// TIA Portal V17 export
// export: Created 2025-03-05T08:00:56.2368358Z, ExportSetting WithDefaults, DisplayName Totally Integrated Automation Portal, DisplayVersion V17 Update 8, DisplayName TIA Portal Openness, DisplayVersion V17 Update 8, DisplayName TIA Portal Version Control Interface, DisplayVersion V17, DisplayName SINAMICS Startdrive Advanced, DisplayVersion V17 SP2, DisplayName SINAMICS Startdrive G110M, G120, G120C, G120D, G120P, G115D, DisplayVersion V17 SP2, DisplayName SINAMICS Startdrive G130, G150, S120, S150, SINAMICS MV, S210, DisplayVersion V17 SP2, DisplayName STEP 7 Professional, DisplayVersion V17 Update 8, DisplayName SINUMERIK ONE STEP 7 Toolbox, DisplayVersion V17 Update 12, DisplayName SINUMERIK 840D sl STEP 7 Toolbox, DisplayVersion V17 Update 12, DisplayName STEP 7 Safety, DisplayVersion V17 Update 6, DisplayName WinCC Advanced, DisplayVersion V17 Update 8
FUNCTION "FC1500_GAS_GENERAL" : Void   // FC1500, LAD
{ S7_Optimized_Access := 'TRUE' }
VERSION : 0.1
// stored: AutoNumber false, IsIECCheckEnabled false, SetENOAutomatically false, UDAEnableTagReadback false
BEGIN

REGION Network 1: CALL FC1501_MAIN_GAS_VALVE
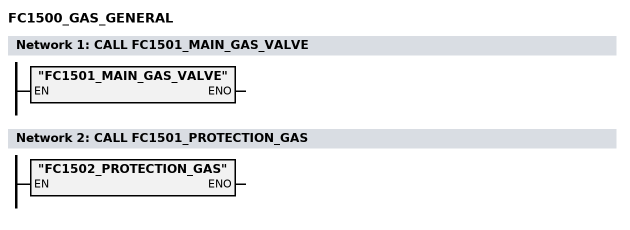
   RUNG wire#powerrail
      "FC1501_MAIN_GAS_VALVE"()
   END_RUNG
   // the same network as SCL:
   "FC1501_MAIN_GAS_VALVE"();
END_REGION

REGION Network 2: CALL FC1501_PROTECTION_GAS
   RUNG wire#powerrail
      "FC1502_PROTECTION_GAS"()
   END_RUNG
   // the same network as SCL:
   "FC1502_PROTECTION_GAS"();
END_REGION
END_FUNCTION
